# EPICS autosave request: leybold/coolpak_settings.req
$(P):HEAD1MODE
$(P):HEAD2MODE
$(P):SYSTEMMODE
